FUNCTION_BLOCK FB_BaseStrategyController
VAR_INPUT
	ambientState : ST_AmbientState;
	
	//actual temperatures in thermal networks
	cnState : ST_BufferStorageState;
	hnltState : ST_BufferStorageState;
END_VAR
VAR_OUTPUT	
	{attribute 'OPC.UA.DA' := '1'}
	cnControl : ST_CoolingNetworkControl;
	{attribute 'OPC.UA.DA' := '1'}	
	hnltControl : ST_LowTemperatureHeatingNetworkControl;
	{attribute 'OPC.UA.DA' := '1'}
	hnltCnLinkageControl : ST_HnltCnLinkageControl;
	
END_VAR
VAR
	//temperature limits for thermal networks
	aTemperatureLimits_HNHT : ARRAY[1..2] OF REAL := [70,90]; //temperature limits for high temperature heating network
	aTemperatureLimits_HNLT : ARRAY[1..2] OF REAL := [30,45]; //temperature limits for low temperature heating network
	aTemperatureLimits_CN : ARRAY[1..2] OF REAL := [5,25]; //temperature limits for cooling network

	//controllers and variables for cooling network
	Controller_eChiller : FB_CTRL_2POINT;
	Controller_eChiller_Parameters : ST_CTRL_2POINT_PARAMS;
	Controller_HVFA_CN : FB_CTRL_2POINT;
	Controller_HVFA_CN_Parameters : ST_CTRL_2POINT_PARAMS;
	
	//controllers and variables for low temperature heating network
	Controller_OuterCapillaryTubeMats : FB_CTRL_2POINT;
	Controller_OuterCapillaryTubeMats_Parameters : ST_CTRL_2POINT_PARAMS;
	
	//controllers and variables for hnlt and cn linkage
	Controller_HeatPump : FB_CTRL_2POINT;
	Controller_HeatPump_Parameters : ST_CTRL_2POINT_PARAMS;	
	Controller_HeatPump_Permission : FB_CTRL_2POINT;
	Controller_HeatPump_Permission_Parameters : ST_CTRL_2POINT_PARAMS;
	
	//clock
	stDefaultParameters_Clock : ST_ClockDefaultParameters := (tTaskCycleTime := GlobalVariables.tCtrlCycleTime_MAIN, tCtrlCycleTime := T#1M);
	Clock : FB_Clock := (ST_DefaultParameters := stDefaultParameters_Clock);
END_VAR

SetTargetTemperatures();
CheckAlgorithmPermission();
AmbientControl();
ControlCN();
ControlHNLT();
ControlHnltCnLinkage();

METHOD AmbientControl : BOOL
VAR_INPUT
END_VAR
//check for heating or cooling mode
IF Clock.stClockState.sintMonth>4 AND Clock.stClockState.sintMonth<10 THEN
	//heating mode
	hnltCnLinkageControl.bHeatingMode := TRUE;
ELSE
	//cooling mode	
	hnltCnLinkageControl.bHeatingMode := FALSE;
END_IF
END_METHOD

METHOD CheckAlgorithmPermission : BOOL
VAR_INPUT
END_VAR
VAR
END_VAR
//check for algorithm permissions
cnControl.bAlgorithmPermission := Limiter(fInput := cnState.fMidTemperature,fLowerLimit := aTemperatureLimits_CN[1],fUpperLimit := aTemperatureLimits_CN[2]);
hnltControl.bAlgorithmPermission := Limiter(fInput := hnltState.fMidTemperature, fLowerLimit := aTemperatureLimits_HNLT[1], fUpperLimit := aTemperatureLimits_HNLT[2]);


//set algorithm permissions to linkage structs
hnltCnLinkageControl.bAlgorithmPermission_CN := cnControl.bAlgorithmPermission;
hnltCnLinkageControl.bAlgorithmPermission_HNLT := hnltControl.bAlgorithmPermission;
END_METHOD

METHOD ControlCN : BOOL
VAR_INPUT
END_VAR
//set hysteresis parameters for two-point controllers in cooling network
Controller_eChiller_Parameters.fHysteresisRange := 4;
Controller_eChiller_Parameters.tCtrlCycleTime := GlobalVariables.tTaskCycleTime_MAIN;
Controller_eChiller_Parameters.tTaskCycleTime := GlobalVariables.tTaskCycleTime_MAIN;

//control strategy for cooling network - fSetpointValue and fActualValue are changed for cooling applications
Controller_eChiller(fSetpointValue := cnState.fMidTemperature,
	fActualValue := cnControl.fTargetTemperature+2,
	eMode := eCTRL_MODE_ACTIVE,
	stParams := Controller_eChiller_Parameters);
cnControl.bSetStatusOn_eChiller := Controller_eChiller.bOut;

//control hvfa storage
//hvfa storage is currently not used
cnControl.bSetStatusOn_HVFASystem := FALSE;
cnControl.bLoading_HVFASystem := FALSE;
END_METHOD

METHOD ControlHNLT : BOOL
VAR_INPUT
END_VAR
//set hysteresis parameters for two-point controllers in cooling network
Controller_OuterCapillaryTubeMats_Parameters.fHysteresisRange := 4;
Controller_OuterCapillaryTubeMats_Parameters.tCtrlCycleTime := GlobalVariables.tTaskCycleTime_MAIN;
Controller_OuterCapillaryTubeMats_Parameters.tTaskCycleTime := GlobalVariables.tTaskCycleTime_MAIN;

//control strategy for cooling network - fSetpointValue and fActualValue are changed for cooling applications
Controller_OuterCapillaryTubeMats(fSetpointValue := hnltState.fMidTemperature,
	fActualValue := aTemperatureLimits_HNLT[2],
	eMode := eCTRL_MODE_ACTIVE,
	stParams := Controller_OuterCapillaryTubeMats_Parameters);
hnltControl.bSetStatusOn_OuterCapillaryTubeMats := Controller_OuterCapillaryTubeMats.bOut;

//control hvfa storage
//hvfa storage is currently not used
hnltControl.bSetStatusOn_HVFASystem := FALSE;
hnltControl.bLoading_HVFASystem := FALSE;
END_METHOD

METHOD ControlHnltCnLinkage : BOOL
VAR_INPUT
END_VAR
//set hysteresis parameters for hnlt cn linkage systems
Controller_HeatPump_Parameters.fHysteresisRange := 4;
Controller_HeatPump_Parameters.tCtrlCycleTime := GlobalVariables.tTaskCycleTime_MAIN;
Controller_HeatPump_Parameters.tTaskCycleTime := GlobalVariables.tTaskCycleTime_MAIN;

Controller_HeatPump_Permission_Parameters.fHysteresisRange := 4;
Controller_HeatPump_Permission_Parameters.tCtrlCycleTime := GlobalVariables.tTaskCycleTime_MAIN;
Controller_HeatPump_Permission_Parameters.tTaskCycleTime := GlobalVariables.tTaskCycleTime_MAIN;

//control heat pump depending on cooling demand in cn
Controller_HeatPump(fSetpointValue := cnState.fUpperTemperature,
	fActualValue := cnControl.fTargetTemperature,
	eMode := eCTRL_MODE_ACTIVE,
	stParams := Controller_HeatPump_Parameters);
	
//control heat pump permission depending on critical temperature in hnlt
Controller_HeatPump_Permission(fSetpointValue := aTemperatureLimits_HNLT[2],
	fActualValue := hnltState.fMidTemperature,
	eMode := eCTRL_MODE_ACTIVE,
	stParams := Controller_HeatPump_Parameters);
	
hnltCnLinkageControl.bSetStatusOn_HeatPump := Controller_HeatPump.bOut AND Controller_HeatPump_Permission.bOut;
END_METHOD

METHOD SetTargetTemperatures : BOOL
VAR_INPUT
END_VAR
//set default target temperatures
cnControl.fTargetTemperature := 15;
hnltControl.fTargetTemperature := 40;

//set target temperatures to linkage structs
hnltCnLinkageControl.fTargetTemperature_CN := cnControl.fTargetTemperature;
hnltCnLinkageControl.fTargetTemperature_HNLT := hnltControl.fTargetTemperature;
hnltCnLinkageControl.fTargetTemperature_ProductionHall := 21;
END_METHOD

END_FUNCTION_BLOCK

(* stored: Version 1.1.0.1, ProductVersion 3.1.4024.10
   POU FB_BaseStrategyController: Id {2cc24fef-e41e-40c1-8491-4b4c0461b6c2}, SpecialFunc None
   Method AmbientControl: Id {259f8bb9-b8e0-4675-99d4-6749b70c4f63}
   Method CheckAlgorithmPermission: Id {66275845-0f5f-4b5e-bd16-5cacbde5e92b}
   Method ControlCN: Id {c114617d-ff2b-491a-a80e-d1c974ffb859}
   Method ControlHNLT: Id {57bcb54f-1f56-4d59-8bc6-dbfcc2a5773d}
   Method ControlHnltCnLinkage: Id {47fe50a8-fa6a-42c9-86f6-4129fa6636fe}
   Method SetTargetTemperatures: Id {6be7450f-8e0b-4497-9741-f2ddcfb682eb} *)
